// TIA Portal V20 export
ORGANIZATION_BLOCK "Main"   // OB1, LAD, ProgramCycle
TITLE = "Main Program Sweep (Cycle)"
{ S7_Optimized_Access := 'TRUE' }
// stored: SetENOAutomatically false
   VAR_INPUT
      Initial_Call : Bool;   // Initial call of this OB
      Remanence : Bool;   // =True, if remanent data are available
   END_VAR
BEGIN

REGION Network 1
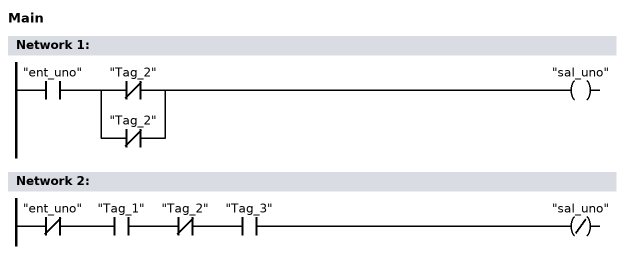
   RUNG wire#powerrail
      Contact( "ent_uno" )
      wire#w1
      I_Contact( "Tag_2" )
      wire#w2
      Coil( "sal_uno" )
   END_RUNG
   RUNG wire#w1
      I_Contact( "Tag_2" )
   END_RUNG wire#w2
   // the same network as SCL:
   "sal_uno" := "ent_uno" AND (NOT "Tag_2" OR NOT "Tag_2");
END_REGION

REGION Network 2
   RUNG wire#powerrail
      I_Contact( "ent_uno" )
      Contact( "Tag_1" )
      I_Contact( "Tag_2" )
      Contact( "Tag_3" )
      I_Coil( "sal_uno" )
   END_RUNG
   // the same network as SCL:
   "sal_uno" := NOT (NOT "ent_uno" AND "Tag_1" AND NOT "Tag_2" AND "Tag_3");
END_REGION
END_ORGANIZATION_BLOCK
